{attribute addProperty BoxType "EK1100-0000-0018"}
{attribute addProperty Id "Beckhoff_EPP1xxxEK1122Beckhoff_EPP1xxxEK1122_CF9B9B855440680"}
{attribute addProperty CRC "2646950657"}
{attribute addProperty SizeInBites "5440"}
{attribute addProperty SizeInBytes "680"}
TYPE Beckhoff_EPP1xxx_9DC54301 EXTENDS EK1100_179A0949 :
STRUCT
	{attribute addProperty Name "Beckhoff_EPP1xxxEK1122"}
	Beckhoff_EPP1xxxEK1122 : Beckhoff_EPP1xxxEK1122_CF9B9B85;
END_STRUCT
END_TYPE

(* stored: Version 1.2.0.0, ProductVersion 3.1.4024.9
   DUT Beckhoff_EPP1xxx_9DC54301: Id {f73ca230-a32a-469c-874b-cd1ba37b35a6} *)
